// TIA Portal V15 export
// export: ExportSetting WithDefaults, WithReadOnly, DisplayName Totally Integrated Automation Portal, DisplayVersion V15, DisplayName TIA Portal Openness, DisplayVersion V15, DisplayName STEP 7 Professional, DisplayVersion V15, DisplayName STEP 7 Safety, DisplayVersion V15, DisplayName WinCC Professional, DisplayVersion V15, DisplayName SIMATIC Visualization Architect, DisplayVersion V15
DATA_BLOCK "ROBNAME"   // DB100
{ S7_Optimized_Access := 'TRUE' }
AUTHOR : INTROSYS
NAME : ROBNAME
VERSION : 0.0
// stored: AutoNumber false, DBAccessibleFromOPCUA true, DownloadWithoutReinit false, InterfaceModifiedDate 2019-04-05T16:56:39.048637Z, IsConsistent true, IsKnowHowProtected false, IsOnlyStoredInLoadMemory false, IsPLCDB false, IsRetainMemResEnabled false, IsWriteProtectedInAS false, MemoryReserve 100, ModifiedDate 2019-04-05T16:57:03.123955Z, ParameterModified 2019-04-05T16:56:39.048637Z, StructureModified 2019-04-05T16:56:39.048637Z
   VAR RETAIN
      Rob { ExternalAccessible := 'False'; ExternalVisible := 'False'; ExternalWritable := 'False'} : "ST_Rob";   // Roboter
      PG { ExternalAccessible := 'False'; ExternalVisible := 'False'; ExternalWritable := 'False'} : "ST_PG";   // Prozessgerätstruktur
      FM { ExternalAccessible := 'False'; ExternalVisible := 'False'; ExternalWritable := 'False'} : Bool;   // Fertigmeldung Gesamt
      K91_Verkl { ExternalAccessible := 'False'; ExternalVisible := 'False'; ExternalWritable := 'False'} : Bool;   // Verklemmanzeige
      Warn { ExternalAccessible := 'False'; ExternalVisible := 'False'; ExternalWritable := 'False'} : Bool;   // Warnung
      Stoe { ExternalAccessible := 'False'; ExternalVisible := 'False'; ExternalWritable := 'False'} : Bool;   // Störung
      Wart { ExternalAccessible := 'False'; ExternalVisible := 'False'; ExternalWritable := 'False'} : Bool;   // Wartung
      PGWarn { ExternalAccessible := 'False'; ExternalVisible := 'False'; ExternalWritable := 'False'} : Bool;   // Warnung
      PGStoe { ExternalAccessible := 'False'; ExternalVisible := 'False'; ExternalWritable := 'False'} : Bool;   // Störung
      PGWart { ExternalAccessible := 'False'; ExternalVisible := 'False'; ExternalWritable := 'False'} : Bool;   // Wartung
      Taktzeit_Plus_Typ { ExternalAccessible := 'False'; ExternalVisible := 'False'; ExternalWritable := 'False'} : Int;   // Uebergabe Typ an FB_Taktzeit_Plus
      TZL_Wert { ExternalAccessible := 'False'; ExternalVisible := 'False'; ExternalWritable := 'False'} : Int;   // Letzter gemesssener diZeitwert in 1/10s
      TZStoe { ExternalAccessible := 'False'; ExternalVisible := 'False'; ExternalWritable := 'False'} : Bool;   // Taktzeit Störung
      TZStop { ExternalAccessible := 'False'; ExternalVisible := 'False'; ExternalWritable := 'False'} : Bool;   // Taktzeit Stopp Hifu
      SFN1 { ExternalAccessible := 'False'; ExternalVisible := 'False'; ExternalWritable := 'False'} : Bool;   // 225050R01SFN1
      Frg_MaschSich { ExternalAccessible := 'False'; ExternalVisible := 'False'; ExternalWritable := 'False'} : Bool;   // Freigabe Maschinensicherheit Hifu
      Frg_MaschSich1 { ExternalAccessible := 'False'; ExternalVisible := 'False'; ExternalWritable := 'False'} : Bool;   // Freigabe Maschinensicherheit Hifu 1
      ExtMedienEIN { ExternalAccessible := 'False'; ExternalVisible := 'False'; ExternalWritable := 'False'} : Bool;   // externe Medien einschalten
      StoeMedien { ExternalAccessible := 'False'; ExternalVisible := 'False'; ExternalWritable := 'False'} : Bool;   // Störung Roboter Medien
      FolgeStart { ExternalAccessible := 'False'; ExternalVisible := 'False'; ExternalWritable := 'False'} : Bool;   // Start Arbeitsfolge Hifu
   END_VAR
BEGIN
END_DATA_BLOCK
